PROGRAM _00_GENERALES
VAR
	Pulso_1s: fbpulse1s;
	
END_VAR

//GENERA PULSOS Y FLANCOS CADA SEGUNDO

Pulso_1s ();

END_PROGRAM

(* stored: Version 1.1.0.1, ProductVersion 3.1.4024.10
   POU _00_GENERALES: Id {636df509-612b-496d-a682-04a085333454}, SpecialFunc None *)
